FUNCTION_BLOCK Getriebemotor
VAR_INPUT
END_VAR
VAR_OUTPUT
END_VAR
VAR
END_VAR

dSub.Q1 := dSub.S8;	// Motor Linkslauf
dSub.Q2 := dSub.S7;	// Motor Rechtslauf
dSub.P1 := dSub.S1;	
dSub.P2 := dSub.S4;
dSub.P3 := dSub.S3;
dSub.P4 := dSub.S6;

END_FUNCTION_BLOCK

(* stored: Version 1.1.0.1, ProductVersion 3.1.4022.7
   POU Getriebemotor: Id {cb65ceda-4bf1-470d-b57d-3c08e6479214}, SpecialFunc None *)
